Fanuc KAREL source: kd00002.KL

-- PROVISIONAL review KL for V1013-1; original PC SHA256 4ec5ca64aee5655e8cf4b613a6ac2ac6a06fce300810f7e490255df06f748ec0
-- Incomplete behavior may be omitted. Consult companion uncertainty JSON. Do not deploy.
PROGRAM KD00002
%NOLOCKGROUP
VAR
  I : INTEGER
  J : INTEGER
  B : BOOLEAN
  R : REAL
  S : STRING[80]
BEGIN
  -- UNRESOLVED_PC offsets 5-12; opcodes 9D,23
  -- UNRESOLVED_PC offsets 17-21; opcodes 7F
END KD00002
